(* PLC project Untitled1, Beckhoff Automation GmbH TF6420 Database Server Query Analyser 1.0.0.0 *)
(* stored: creationDateTime 2022-01-14T14:12:53, modificationDateTime 2022-01-14T14:12:53 *)

TYPE ST_SelectStructData : STRUCT
  datetime : STRING(255);
  trailer_id_lead : LINT;
  trailer_id_rear : LINT;
  latitude : REAL;
  longitude : REAL;
  speed : REAL;
  overspeed : LINT;
  payload_lead : REAL;
  payload_rear : REAL;
  overload_lead : LINT;
  overload_rear : LINT;
  pressure_lead : REAL;
  pressure_rear : REAL;
  overpressure_lead : LINT;
  overpressure_rear : LINT;
  event_code : LINT;
END_STRUCT;
END_TYPE
